(* IEC 61131-3 sources: repolevel_ST_code_completion/output/0122完整版本_无planner目前sota/repoeval_three-axis_CNC_motion/readful_result, 4 files *)

(* ---- INIT_CNC_System.st ---- *)
FUNCTION INIT_CNC_System : BOOL
VAR_IN_OUT
	fbSMC_ReadNCFile		:	SMC_ReadNCFile;
	fbSMC_NCDecoder			:	SMC_NCDecoder;
	fbSMC_CheckVelocities	:	SMC_CheckVelocities;
	fbSMC_Interpolator		:	SMC_Interpolator;
	fbSMC_ControlAxisXByPos	:	SMC_ControlAxisByPos;
	fbSMC_ControlAxisYByPos	:	SMC_ControlAxisByPos;
	fbSMC_ControlAxisZByPos	:	SMC_ControlAxisByPos;
	fbSMC_AXISX_HOMING		:	SMC_HOMING;
	fbSMC_AXISY_HOMING		:	SMC_HOMING;
	fbSMC_AXISZ_HOMING		:	SMC_HOMING;
	fbMC_AXISX_STOP			:	MC_STOP;
	fbMC_AXISY_STOP			:	MC_STOP;
	fbMC_AXISZ_STOP			:	MC_STOP;
END_VAR
VAR_INPUT
	AxisX					:	SM3_Basic.AXIS_REF_SM3
	AxisY					:	SM3_Basic.AXIS_REF_SM3
	AxisZ					:	SM3_Basic.AXIS_REF_SM3
END_VAR
VAR
    bInitSuccess : BOOL;
END_VAR

fbSMC_ReadNCFile(bExecute := FALSE);
fbSMC_NCDecoder(bExecute := FALSE, ncprog := fbSMC_ReadNCFile.ncprog);
fbSMC_CheckVelocities(bExecute := FALSE);
fbSMC_Interpolator(bExecute := FALSE);

fbSMC_AXISX_HOMING(bExecute := FALSE, Axis := AxisX);
fbSMC_AXISY_HOMING(bExecute := FALSE, Axis := AxisY);
fbSMC_AXISZ_HOMING(bExecute := FALSE, Axis := AxisZ);

fbMC_AXISX_STOP(bExecute := FALSE, Axis := AxisX);
fbMC_AXISY_STOP(bExecute := FALSE, Axis := AxisY);
fbMC_AXISZ_STOP(bExecute := FALSE, Axis := AxisZ);

bInitSuccess := TRUE;
RETURN bInitSuccess;
END_FUNCTION

(* ---- FB_TripleAxisHoming.st ---- *)
FUNCTION_BLOCK FB_TripleAxisHoming
VAR_INPUT
	bExecute			:	BOOL;				//执行回零信号
	AxisX				:	AXIS_REF;			//X轴引用
	AxisY				:	AXIS_REF;			//Y轴引用
	AxisZ				:	AXIS_REF;			//Z轴引用
	bAxisXRefSwitch		:	BOOL;				//X轴零点开关
	bAxisYRefSwitch		:	BOOL;				//Y轴零点开关
	bAxisZRefSwitch		:	BOOL;				//Z轴零点开关
	fVelocitySlow		:	REAL;				//慢速回零速度
	fVelocityFast		:	REAL;				//快速回零速度
	fAcceleration		:	REAL;				//加速度
	fDeceleration		:	REAL;				//减速度
END_VAR
VAR_OUTPUT
	bHomeOK				:	BOOL;				//三轴都回零完成
	bAxisXHomeOK		:	BOOL;				//X轴回零完成
	bAxisYHomeOK		:	BOOL;				//Y轴回零完成
	bAxisZHomeOK		:	BOOL;				//Z轴回零完成
	bBusy				:	BOOL;				//回零进行中
	bError				:	BOOL;				//错误标志
	sErrorString		:	STRING;				//错误信息字符串
END_VAR
VAR
	fbHomingX			:	SMC_HOMING;			//X轴回零功能块
	fbHomingY			:	SMC_HOMING;			//Y轴回零功能块
	fbHomingZ			:	SMC_HOMING;			//Z轴回零功能块
	bXHomingDone		:	BOOL;				//X轴回零完成标志
	bYHomingDone		:	BOOL;				//Y轴回零完成标志
	bZHomingDone		:	BOOL;				//Z轴回零完成标志
	bXHomingError		:	BOOL;				//X轴回零错误标志
	bYHomingError		:	BOOL;				//Y轴回零错误标志
	bZHomingError		:	BOOL;				//Z轴回零错误标志
	sTempErrorString	:	STRING;				//临时错误信息字符串
END_VAR

IF bExecute THEN
	bBusy := TRUE;
	bError := FALSE;
	sErrorString := '';

	// X轴回零过程
	fbHomingX.Axis := AxisX;
	fbHomingX.Execute := NOT bXHomingDone;
	fbHomingX.Velocity := fVelocityFast;
	fbHomingX.Acceleration := fAcceleration;
	fbHomingX.Deceleration := fDeceleration;
	fbHomingX.HomeSwitch := bAxisXRefSwitch;
	fbHomingX();
	bXHomingDone := fbHomingX.Done;
	bXHomingError := fbHomingX.Error;

	// Y轴回零过程
	fbHomingY.Axis := AxisY;
	fbHomingY.Execute := NOT bYHomingDone AND bXHomingDone;
	fbHomingY.Velocity := fVelocityFast;
	fbHomingY.Acceleration := fAcceleration;
	fbHomingY.Deceleration := fDeceleration;
	fbHomingY.HomeSwitch := bAxisYRefSwitch;
	fbHomingY();
	bYHomingDone := fbHomingY.Done;
	bYHomingError := fbHomingY.Error;

	// Z轴回零过程
	fbHomingZ.Axis := AxisZ;
	fbHomingZ.Execute := NOT bZHomingDone AND bYHomingDone;
	fbHomingZ.Velocity := fVelocityFast;
	fbHomingZ.Acceleration := fAcceleration;
	fbHomingZ.Deceleration := fDeceleration;
	fbHomingZ.HomeSwitch := bAxisZRefSwitch;
	fbHomingZ();
	bZHomingDone := fbHomingZ.Done;
	bZHomingError := fbHomingZ.Error;

	// 错误处理
	IF bXHomingError THEN
		bError := TRUE;
		sTempErrorString := fbHomingX.ErrorID;
	ELSIF bYHomingError THEN
		bError := TRUE;
		sTempErrorString := fbHomingY.ErrorID;
	ELSIF bZHomingError THEN
		bError := TRUE;
		sTempErrorString := fbHomingZ.ErrorID;
	END_IF;

	IF bError THEN
		sErrorString := CONCAT('Homing Error: ', sTempErrorString);
		bBusy := FALSE;
		RETURN;
	END_IF;

	// 回零完成状态
	bAxisXHomeOK := bXHomingDone;
	bAxisYHomeOK := bYHomingDone;
	bAxisZHomeOK := bZHomingDone;
	bHomeOK := bXHomingDone AND bYHomingDone AND bZHomingDone;

	IF bHomeOK THEN
		bBusy := FALSE;
	END_IF;
ELSE
	bBusy := FALSE;
	bHomeOK := FALSE;
	bAxisXHomeOK := FALSE;
	bAxisYHomeOK := FALSE;
	bAxisZHomeOK := FALSE;
	bError := FALSE;
	sErrorString := '';
END_IF;
END_FUNCTION_BLOCK

(* ---- FB_TripleAxisPower.st ---- *)
FUNCTION_BLOCK FB_TripleAxisPower
VAR_INPUT
	AxisX			:	SM3_Basic.AXIS_REF_SM3			//X轴引用
	AxisY			:	SM3_Basic.AXIS_REF_SM3			//Y轴引用
	AxisZ			:	SM3_Basic.AXIS_REF_SM3			//Z轴引用
	bServoEnable	:	BOOL;				//伺服使能信号
END_VAR
VAR_OUTPUT
	bReady			:	BOOL;				//三轴都准备就绪
	bAxisXReady		:	BOOL;				//X轴准备就绪
	bAxisYReady		:	BOOL;				//Y轴准备就绪
	bAxisZReady		:	BOOL;				//Z轴准备就绪
	bError			:	BOOL;				//错误标志
	sErrorString	:	STRING;				//错误信息字符串
END_VAR
VAR
	fbPowerX		:	MC_POWER;			//X轴电源控制
	fbPowerY		:	MC_POWER;			//Y轴电源控制
	fbPowerZ		:	MC_POWER;			//Z轴电源控制
	bErrorX			:	BOOL;				//X轴错误标志
	bErrorY			:	BOOL;				//Y轴错误标志
	bErrorZ			:	BOOL;				//Z轴错误标志
	sErrorX			:	STRING;				//X轴错误信息
	sErrorY			:	STRING;				//Y轴错误信息
	sErrorZ			:	STRING;				//Z轴错误信息
END_VAR

fbPowerX(
	Enable := bServoEnable,
	bRegulatorOn := bServoEnable,
	bDriveStart := bServoEnable,
	Axis := AxisX
);

fbPowerY(
	Enable := bServoEnable,
	bRegulatorOn := bServoEnable,
	bDriveStart := bServoEnable,
	Axis := AxisY
);

fbPowerZ(
	Enable := bServoEnable,
	bRegulatorOn := bServoEnable,
	bDriveStart := bServoEnable,
	Axis := AxisZ
);

bAxisXReady := fbPowerX.Status = MC_POWER_STATUS.PowerOn;
bAxisYReady := fbPowerY.Status = MC_POWER_STATUS.PowerOn;
bAxisZReady := fbPowerZ.Status = MC_POWER_STATUS.PowerOn;

bErrorX := fbPowerX.Error;
bErrorY := fbPowerY.Error;
bErrorZ := fbPowerZ.Error;

sErrorX := fbPowerX.ErrorID;
sErrorY := fbPowerY.ErrorID;
sErrorZ := fbPowerZ.ErrorID;

bError := bErrorX OR bErrorY OR bErrorZ;

IF bError THEN
	IF bErrorX THEN
		sErrorString := 'X Axis Error: ' + sErrorX;
	ELSIF bErrorY THEN
		sErrorString := 'Y Axis Error: ' + sErrorY;
	ELSIF bErrorZ THEN
		sErrorString := 'Z Axis Error: ' + sErrorZ;
	END_IF;
ELSE
	sErrorString := '';
END_IF;

bReady := bAxisXReady AND bAxisYReady AND bAxisZReady;
END_FUNCTION_BLOCK

(* ---- FB_TripleAxisStop.st ---- *)
FUNCTION_BLOCK FB_TripleAxisStop
VAR_INPUT
	AxisX			:	SM3_Basic.AXIS_REF_SM3			//X轴引用
	AxisY			:	SM3_Basic.AXIS_REF_SM3			//Y轴引用
	AxisZ			:	SM3_Basic.AXIS_REF_SM3			//Z轴引用
	bExecute		:	BOOL;				//执行停止信号
	rDeceleration	:	REAL := 100.0;		//减速度
END_VAR
VAR_OUTPUT
	bDone			:	BOOL;				//三轴都停止完成
	bBusy			:	BOOL;				//停止进行中
	bError			:	BOOL;				//错误标志
	sErrorString	:	STRING;				//错误信息字符串
END_VAR
VAR
	fbStopX			:	MC_STOP;			//X轴停止
	fbStopY			:	MC_STOP;			//Y轴停止
	fbStopZ			:	MC_STOP;			//Z轴停止
	bStopXDone		:	BOOL;				//X轴停止完成
	bStopYDone		:	BOOL;				//Y轴停止完成
	bStopZDone		:	BOOL;				//Z轴停止完成
	bStopXError		:	BOOL;				//X轴停止错误
	bStopYError		:	BOOL;				//Y轴停止错误
	bStopZError		:	BOOL;				//Z轴停止错误
	sStopXErrorString:	STRING;				//X轴错误信息
	sStopYErrorString:	STRING;				//Y轴错误信息
	sStopZErrorString:	STRING;				//Z轴错误信息
END_VAR

fbStopX(
	Execute := bExecute,
	Deceleration := rDeceleration,
	Axis := AxisX
);
bStopXDone := fbStopX.Done;
bStopXError := fbStopX.Error;
sStopXErrorString := fbStopX.ErrorID;

fbStopY(
	Execute := bExecute,
	Deceleration := rDeceleration,
	Axis := AxisY
);
bStopYDone := fbStopY.Done;
bStopYError := fbStopY.Error;
sStopYErrorString := fbStopY.ErrorID;

fbStopZ(
	Execute := bExecute,
	Deceleration := rDeceleration,
	Axis := AxisZ
);
bStopZDone := fbStopZ.Done;
bStopZError := fbStopZ.Error;
sStopZErrorString := fbStopZ.ErrorID;

bDone := bStopXDone AND bStopYDone AND bStopZDone;
bBusy := NOT bDone;
bError := bStopXError OR bStopYError OR bStopZError;

IF bStopXError THEN
	sErrorString := sStopXErrorString;
ELSIF bStopYError THEN
	sErrorString := sStopYErrorString;
ELSIF bStopZError THEN
	sErrorString := sStopZErrorString;
ELSE
	sErrorString := '';
END_IF;
END_FUNCTION_BLOCK
